// TIA Portal V19 export
TYPE "Positioning_MOL_Machine_Par"
// stored: Access Published
   STRUCT
      PosTolerance { S7_SetPoint := 'True'} : LReal;
      DelayInPosition { S7_SetPoint := 'True'} : Time;
      Minus_Limit { S7_SetPoint := 'True'} : LReal;
      Plus_Limit { S7_SetPoint := 'True'} : LReal;
      PreCutOff { S7_SetPoint := 'True'} : LReal;
   END_STRUCT;
END_TYPE
